Yaskawa INFORM job: INIT_ROS.JBI

/JOB
//NAME INIT_ROS
//POS
///NPOS 0,0,0,0,0,0
//INST
///DATE 2014/06/16 09:29
///ATTR SC,RW
NOP
PSTART JOB:ROS_R1 SUB1
PSTART JOB:ROS_S1 SUB2
PWAIT SUB1
END
